ABB RobotStudio station: Lab12_ex1.rsstnx

Station Lab12_ex1 (saved by RobotStudio 23.3.10550.0)
Controller Controller1
  mechanical unit ROB_1: IRB4600_20_250_C_01, 6 joints, base frame (0, 0, 0) mm
  mechanical unit ROB_2: IRB2400_10_150__02, 6 joints, base frame (3142.23, 0, 0) mm, rotated rx 0 ry 0 rz 180 deg
Layout (positions relative to the parent item):
  - IRB4600_20_250_C_01 [mechanism, from %ABB.RobotStudio.Models.IRB4600%\IRB4600_20_250_C_G_01.rslib] at (0, 0, 0) mm; joint values [-0.4165, -0.1445, 0.1779, 0, 0.4902, 0] (rad or m)
  - IRB2400_10_150__02 [mechanism, from %ABB.RobotStudio.Models.IRB2400%\IRB2400_10_150_G_02.rslib] at (3142.23, 0, 0) mm, rotated rx 0 ry 0 rz 180 deg; joint values [-0.8041, 0, 0, 0, 0.5236, 0] (rad or m)
